// TwinCAT 3 PLC project AW_PLC
// ProgramVersion: 3.1.4023.0
// libraries:
//   Tc2_EtherCAT, * (Beckhoff Automation GmbH)
//   Tc2_Standard, * (Beckhoff Automation GmbH)
//   Tc2_System, * (Beckhoff Automation GmbH)
//   Tc3_Module, * (Beckhoff Automation GmbH)
// project tree:
//   DUTs/ TextList.TcTLO
//   / Gestore di visualizzazione.TcVMO (not stored), GlobalTextList.TcGTLO, PlcTask.TcTTO, Sfondo.TcIPO (not stored)
//   GVLs/ CONST.TcGVL, CTRL.TcGVL, ENC.TcGVL, MODE.TcGVL, MOTOR.TcGVL, PLC_ERROR.TcGVL, TRAJ.TcGVL
//   POUs/ HMI.TcPOU, INIT.TcPOU, MAIN.TcPOU, SDO.TcPOU, STATE_MACHINE.TcPOU
//   POUs/Modes/ Cyclic_sync_pos.TcPOU, Cyclic_sync_torq.TcPOU, Cyclic_sync_vel.TcPOU, Position_profile.TcPOU, Torque_profile.TcPOU, Velocity_profile.TcPOU
//   POUs/Trajectories/ BWPoly3.TcPOU, BWPoly4.TcPOU, BWPoly5.TcPOU, FWPoly3.TcPOU, FWPoly4.TcPOU, FWPoly5.TcPOU
//   VISUs/ ControlPanel.TcVIS

CONFIGURATION AW_PLC
    RESOURCE PLC ON TwinCAT3
        TASK PlcTask(INTERVAL := T#1ms, PRIORITY := 20);
        PROGRAM MAIN WITH PlcTask : MAIN;
    END_RESOURCE
END_CONFIGURATION

// ---- GVLs/CONST.TcGVL
{attribute 'qualified_only'}
VAR_GLOBAL CONSTANT
	
END_VAR
VAR_GLOBAL CONSTANT
	PI_2_MIL: DINT := 6283185;
	COUNT: DINT := 1048576;
END_VAR

// ---- GVLs/CTRL.TcGVL
{attribute 'qualified_only'}
VAR_GLOBAL
	state_axis: INT;
	working_counter_status AT %I*: BYTE;
	error AT %I*: INT;
	start					: BOOL := FALSE; 		// Start al movimento
	stop					: BOOL := FALSE;		// Stop al movimento
	opmode AT%Q*		 	: SINT := 8; 			// Modo operativo
	in_opmode AT%I* 		: SINT; 				// Modo operativo letto da giunto
	status_word AT %I*: UINT;
	control_word AT %Q*: UINT;
	sdo: BOOL := FALSE;
	a: BOOL := TRUE;
	b: BOOL;
	read_error: BOOL;
	set_up: BOOL := TRUE;
	wait: BOOL := TRUE;
	active: BOOL := TRUE;
END_VAR

// ---- GVLs/ENC.TcGVL
{attribute 'qualified_only'}
VAR_GLOBAL
		// Approssimato da 2^20/360
	DEG_TO_INC: DINT := 2912;
	RPM_TO_INCS: DINT := 17476;
END_VAR

// ---- GVLs/MODE.TcGVL
{attribute 'qualified_only'}
VAR_GLOBAL CONSTANT
	PROFILE_POSITION	: SINT := 1;
	PROFILE_VELOCITY	: SINT := 3;
	TORQUE_PROFILE		: SINT := 4;
	CYCLIC_SYNC_POS		: SINT := 8;
	CYCLIC_SYNC_VEL		: SINT := 9;
	CYCLIC_SYNC_TORQ	: SINT := 10;
END_VAR

// ---- GVLs/MOTOR.TcGVL
{attribute 'qualified_only'}
VAR_GLOBAL
END_VAR
VAR_GLOBAL
	GEAR_RATIO				: DINT 	:= 51;
	NOMINAL_CURRENT			: INT 	:= 38;	// [A]
	TORQUE_CONSTANT			: INT 	:= 115; // [mNm/A]
	actual_vel_rpm AT %I*			: DINT;		// 
	// In per thousand of the nominal torque
	actual_torque AT %I*			: INT;
	actual_pos_inc AT %I*	: DINT; 		// Posizione reale [cnt]
	RATED_TORQUE_NM: LREAL := 3;
	RATED_SPEED_RPM: UDINT := 1400;
END_VAR

// ---- GVLs/PLC_ERROR.TcGVL
{attribute 'qualified_only'}
VAR_GLOBAL CONSTANT
END_VAR
VAR_GLOBAL CONSTANT
	TRAJ_NO_SETUP: UINT := 1;
	MODE_NO_SETUP: INT := 2;
END_VAR

// ---- GVLs/TRAJ.TcGVL
{attribute 'qualified_only'}
VAR_GLOBAL
	end_pos_inc					: DINT := 0; 		// Posizione finale
	target_pos_inc AT %Q* 	: DINT; 			// Posizione target [cnt]
	// Velocità target [cnt]
	target_vel_mrpm AT %Q*	: DINT;
	start_pos_inc				: DINT := 0; 		// Posizione di start
	tempo					: LREAL := 0; 		// tempo [ms]
	offset_inc: DINT;
	periodo_ms					: LREAL := 1; 		// Durata poly5 [s]	
	delta_t					: LREAL; 			// Delta t per ogni ciclo
	v_max_incs					: DINT; 	// Velocità massima raggiungibile 
	status: BOOL := 0;
	error: UINT := 0;
	v_max_rpm_low: LREAL;
	
	position_selector_deg				: DINT := 180; 	// Offset posizione poly5 [deg]
	target_torque_per_thousand AT %Q*: INT;
	speed_selector_rpm					: UDINT := 500; 	// Velocità massima raggiungibile a freddo 1600 [rpm]
	// [Nm]
	torque_selector_Nm: LREAL := 0.40;
	speed_demand_value AT %I*: DINT;
END_VAR

// ---- POUs/MAIN.TcPOU
PROGRAM MAIN

HMI();
SDO();
STATE_MACHINE();

END_PROGRAM

// ---- POUs/HMI.TcPOU
PROGRAM HMI
VAR
	no_ecat_light: BOOL;
	error_light: BOOL;
	reset_button: BOOL;
	actual_speed_rpm: LREAL;
	actual_torque_nm_fast: LREAL;
	actual_torque_nm_slow: LREAL;
	target_error: DINT;
	count: UDINT := 0;
	status_light: BOOL;
	reset_light: BOOL;
	out_limits_light: BOOL;
	error_output: STRING;
	start_light: BOOL := FALSE;
END_VAR

IF(count = 100)THEN
	//Errors Manage
	IF((CTRL.status_word AND 16#0F)= 16#8)THEN
		error_light := TRUE;
		CTRL.read_error := TRUE;
		IF(CTRL.status_word = 16#B8)THEN
			reset_light		:= TRUE;
		END_IF
		IF(CTRL.status_word = 16#1038)THEN
			out_limits_light	:= TRUE;
		ELSE
			out_limits_light	:= FALSE;
		END_IF
	END_IF
	
	IF (CTRL.working_counter_status = 0) THEN
		no_ecat_light := FALSE;
	ELSE
		no_ecat_light := TRUE;
	END_IF
	
	IF(STATE_MACHINE.timer.Q)THEN 
		CTRL.wait := FALSE;
	ELSE
		CTRL.wait := TRUE;
	END_IF
	
	IF (NOT(CTRL.error = 0 AND TRAJ.error = 0)) THEN 
		error_light := TRUE;
	ELSE
		error_light := FALSE;
	END_IF
	
	IF(CTRL.status_word.0 = 0)THEN
		status_light := FALSE;
		CTRL.read_error := TRUE;
	ELSE
		status_light := TRUE;
		CTRL.read_error := FALSE;	
	END_IF
	
	//Buttons manager
	IF (reset_button) THEN
		STATE_MACHINE.timer(IN:=FALSE);
		CTRL.state_axis	:= 0;
		CTRL.error		:= 0;
		CTRL.control_word := 16#80;
		CTRL.sdo		:= FALSE;
		error_light 	:= FALSE;
		reset_light		:= FALSE;
		out_limits_light:= FALSE;
		reset_button 	:= FALSE;
	END_IF
	
	IF(CTRL.set_up = FALSE)THEN
		INIT();
		CTRL.state_axis	:= 0;
		CTRL.active 	:= TRUE;
	ELSE
		CTRL.active 	:= FALSE;	
	END_IF
		
	//Updates
	actual_speed_rpm		:= MOTOR.actual_vel_rpm*MOTOR.GEAR_RATIO/1000;	
	actual_torque_nm_fast 	:= (MOTOR.actual_torque * MOTOR.RATED_TORQUE_NM)/1000;
	actual_torque_nm_slow 	:= actual_torque_nm_fast * DINT_TO_LREAL(MOTOR.GEAR_RATIO);
	
	count := 0;
ELSE
	count:= count + 1;
END_IF

END_PROGRAM

// ---- POUs/STATE_MACHINE.TcPOU
PROGRAM STATE_MACHINE
VAR
	timer: TON;
END_VAR

IF ( CTRL.sdo = TRUE)THEN
	timer(IN:=TRUE);
	IF (timer.Q = TRUE) THEN
		CASE CTRL.in_opmode OF
			MODE.PROFILE_POSITION:
				Position_profile();	
			MODE.PROFILE_VELOCITY:
				Velocity_profile();
			MODE.TORQUE_PROFILE:
				Torque_profile();
			MODE.CYCLIC_SYNC_POS:
				Cyclic_sync_pos();
			MODE.CYCLIC_SYNC_VEL:
				Cyclic_sync_vel();
			MODE.CYCLIC_SYNC_TORQ:
				Cyclic_sync_torq();	
		ELSE
			CTRL.error:= PLC_ERROR.MODE_NO_SETUP;		
		END_CASE	
	END_IF
END_IF

END_PROGRAM

// ---- POUs/SDO.TcPOU
PROGRAM SDO
VAR
	
	userNetId             	: T_AmsNetId 		:= '192.168.12.90.4.1'; 	// Have to be entered
   	userSlaveAddr         	: UINT 				:= 1001;     				// Have to be entered
	//CoE reading 
	fb_coe_read1           	: FB_EcCoESdoRead;  						// Function Block for reading from CoE
	fb_coe_read2           	: FB_EcCoESdoRead;
	fb_coe_read3           	: FB_EcCoESdoRead;
	fb_coe_read4           	: FB_EcCoESdoRead;
	fb_coe_read5           	: FB_EcCoESdoRead;
	fb_coe_read6           	: FB_EcCoESdoRead;
	fb_coe_read7           	: FB_EcCoESdoRead;
	fb_coe_read8           	: FB_EcCoESdoRead;
	
	fb_coe_write1           : FB_EcCoESdoWrite;
	fb_coe_write2           : FB_EcCoESdoWrite;
	fb_coe_write3           : FB_EcCoESdoWrite;
	fb_coe_write4           : FB_EcCoESdoWrite;
	fb_coe_write5           : FB_EcCoESdoWrite;
	fb_coe_write6           : FB_EcCoESdoWrite;
	fb_coe_write7           : FB_EcCoESdoWrite;
	fb_coe_write8           : FB_EcCoESdoWrite;
	fb_coe_write9           : FB_EcCoESdoWrite;
	fb_coe_write10          : FB_EcCoESdoWrite;
	fb_coe_write11          : FB_EcCoESdoWrite;
	fb_coe_write12          : FB_EcCoESdoWrite;
	fb_coe_write13          : FB_EcCoESdoWrite;
	fb_coe_write14          : FB_EcCoESdoWrite;
	
	motor_revolutions		: UDINT;
	shaft_revolutions		: UDINT;
	enc_resolution			: UDINT := 1048576;
	motor_rated_torque		: DINT;
	max_motor_speed			: UDINT;	
	
	profile_velocity		: UDINT := 0;
	profile_acceleration	: UDINT := 20000;
	profile_deceleration	: UDINT := 20000;
	quick_stop_deceleration	: UDINT := 10000;
	position_window			: UDINT := 100;
	velocity_window			: UINT := 500;
	velocity_window_time	: UINT := 0;
	torque_window			: UINT := 100;
	torque_window_time		: UINT := 0;
	torque_slope			: UDINT := 100;
	written_speed			: UDINT;
	count: INT := 0;
	bExecuteworld: BOOL := FALSE;
	error_report: STRING;
	position_filter_type: USINT := 1;
	position_filter_frequency: UDINT := 200;
	r_position_filter_type: USINT;
	r_position_filter_frequency: UDINT;
	velocity_filter_type: USINT := 1;
	velocity_filter_frequency: UDINT := 100;
END_VAR

//****************** SDO *****************
IF (CTRL.read_error = TRUE) THEN
	fb_coe_read6(bExecute := FALSE);
	fb_coe_read6(
			sNetId		:= userNetId, 
			nSlaveAddr	:= userSlaveAddr, 
			nSubIndex	:= 1, 
			nIndex		:= 16#203F,
			pDstBuf		:= ADR(error_report), 
			cbBufLen    := SIZEOF(error_report), 
			bExecute    := TRUE, 
			tTimeout    := T#1S);
	CTRL.read_error := FALSE;
END_IF

IF (CTRL.sdo = FALSE AND HMI.error_light = FALSE)  THEN

    // read
	IF ( count = 0 ) THEN
		fb_coe_read1(bExecute := FALSE);
		fb_coe_read2(bExecute := FALSE);
		fb_coe_read3(bExecute := FALSE);
		fb_coe_read4(bExecute := FALSE);
		fb_coe_read5(bExecute := FALSE);
		fb_coe_write1(bExecute := FALSE);
		fb_coe_write2(bExecute := FALSE);
		fb_coe_write3(bExecute := FALSE);
		fb_coe_write4(bExecute := FALSE);
		fb_coe_write5(bExecute := FALSE);
		fb_coe_write6(bExecute := FALSE);
		fb_coe_write7(bExecute := FALSE);
		fb_coe_write8(bExecute := FALSE);
		fb_coe_write9(bExecute := FALSE);
		fb_coe_write10(bExecute := FALSE);
		fb_coe_write11(bExecute := FALSE);
		fb_coe_write12(bExecute := FALSE);
		fb_coe_write13(bExecute := FALSE);
		fb_coe_write14(bExecute := FALSE);
		count := count +1;
		STATE_MACHINE.timer(IN:=FALSE,PT:=T#4S);
	END_IF

	
	IF ( NOT bExecuteworld AND count = 1) THEN
		fb_coe_read1(
			sNetId        := userNetId, 
			nSlaveAddr    := userSlaveAddr, 
			nSubIndex    := 1, 
			nIndex        := 16#6091,
			pDstBuf        := ADR(motor_revolutions), 
			cbBufLen    := SIZEOF(motor_revolutions), 
			bExecute    := TRUE, 
			tTimeout    := T#1S);
	
		IF (NOT fb_coe_read1.bBusy) THEN
			bExecuteworld := FALSE;
			fb_coe_read1(bExecute := FALSE);
			count := count + 1;
		END_IF
		
	END_IF
	IF ( NOT bExecuteworld AND count = 2) THEN
		fb_coe_read2(
			sNetId        := userNetId, 
			nSlaveAddr    := userSlaveAddr, 
			nSubIndex    := 2, 
			nIndex        := 16#6091,
			pDstBuf     := ADR(shaft_revolutions), 
			cbBufLen    := SIZEOF(shaft_revolutions), 
			bExecute    := TRUE, 
			tTimeout    := T#1S);	
			
		IF (NOT fb_coe_read2.bBusy) THEN
			bExecuteworld := FALSE;
			fb_coe_read2(bExecute := FALSE);
			count := count + 1;
		END_IF
		
	END_IF
	IF ( NOT bExecuteworld AND count = 3) THEN
		fb_coe_read3(
			sNetId        := userNetId, 
			nSlaveAddr    := userSlaveAddr, 
			nSubIndex    := 3, 
			nIndex        := 16#2110,
			pDstBuf        := ADR(enc_resolution), 
			cbBufLen    := SIZEOF(enc_resolution), 
			bExecute    := TRUE, 
			tTimeout    := T#1S);
	
		IF (NOT fb_coe_read3.bBusy) THEN
			bExecuteworld := FALSE;
			fb_coe_read3(bExecute := FALSE);
			count := count + 1;
		END_IF
		
	END_IF
	IF ( NOT bExecuteworld AND count = 4) THEN
		fb_coe_read4(
			sNetId      := userNetId, 
			nSlaveAddr  := userSlaveAddr, 
			nSubIndex   := 0, 
			nIndex      := 16#6076,
			pDstBuf     := ADR(motor_rated_torque), 
			cbBufLen    := SIZEOF(motor_rated_torque), 
			bExecute    := TRUE, 
			tTimeout    := T#1S);
		IF (NOT fb_coe_read4.bBusy) THEN
			bExecuteworld := FALSE;
			fb_coe_read4(bExecute := FALSE);
			count := count + 1;
		END_IF
		
	END_IF
	IF ( NOT bExecuteworld AND count = 5) THEN
		fb_coe_read5(
			sNetId      := userNetId, 
			nSlaveAddr  := userSlaveAddr, 
			nSubIndex   := 0, 
			nIndex      := 16#6080,
			pDstBuf     := ADR(max_motor_speed), 
			cbBufLen    := SIZEOF(max_motor_speed), 
			bExecute    := TRUE, 
			tTimeout    := T#1S);
		IF (NOT fb_coe_read5.bBusy) THEN
			bExecuteworld := FALSE;
			fb_coe_read5(bExecute := FALSE);
			count := count + 1;
		END_IF
	END_IF
	IF ( NOT bExecuteworld AND count = 6) THEN
		fb_coe_read7(
			sNetId      := userNetId, 
			nSlaveAddr  := userSlaveAddr, 
			nSubIndex   := 1, 
			nIndex      := 16#2022,
			pDstBuf     := ADR(r_position_filter_type), 
			cbBufLen    := SIZEOF(r_position_filter_type), 
			bExecute    := TRUE, 
			tTimeout    := T#1S);
		IF (NOT fb_coe_read7.bBusy) THEN
			bExecuteworld := FALSE;
			fb_coe_read7(bExecute := FALSE);
			count := count + 1;
		END_IF
	END_IF
	IF ( NOT bExecuteworld AND count = 7) THEN
		fb_coe_read8(
			sNetId      := userNetId, 
			nSlaveAddr  := userSlaveAddr, 
			nSubIndex   := 2, 
			nIndex      := 16#2022,
			pDstBuf     := ADR(r_position_filter_frequency), 
			cbBufLen    := SIZEOF(r_position_filter_frequency), 
			bExecute    := TRUE, 
			tTimeout    := T#1S);
		IF (NOT fb_coe_read8.bBusy) THEN
			bExecuteworld := FALSE;
			fb_coe_read8(bExecute := FALSE);
			count := count + 1;
		END_IF
	END_IF
	
    //write
	
	IF ( NOT bExecuteworld AND count = 8) THEN
		//defined by user panel
		profile_velocity 	:= TRAJ.speed_selector_rpm * 1000/DINT_TO_UDINT(MOTOR.GEAR_RATIO);
		fb_coe_write1(
			sNetId     := userNetId,
			nSlaveAddr := userSlaveAddr,
			nIndex     := 16#6081,
			nSubIndex  := 0,
			pSrcBuf    := ADR(profile_velocity),
			cbBufLen   := SIZEOF(profile_velocity),
			bExecute   := TRUE);
		IF (NOT fb_coe_write1.bBusy) THEN
			bExecuteworld := FALSE;
			fb_coe_write1(bExecute := FALSE);
			count := count + 1;
		END_IF
	END_IF
	IF ( NOT bExecuteworld AND count = 9) THEN
		fb_coe_write2(
			sNetId     := userNetId,
			nSlaveAddr := userSlaveAddr,
			nIndex     := 16#6083,
			nSubIndex  := 0,
			pSrcBuf    := ADR(profile_acceleration),
			cbBufLen   := SIZEOF(profile_acceleration),
			bExecute   := TRUE);
		IF (NOT fb_coe_write2.bBusy) THEN
			bExecuteworld := FALSE;
			fb_coe_write2(bExecute := FALSE);
			count := count + 1;
		END_IF
	END_IF
	IF ( NOT bExecuteworld AND count = 10) THEN
		fb_coe_write3(
			sNetId     := userNetId,
			nSlaveAddr := userSlaveAddr,
			nIndex     := 16#6084,
			nSubIndex  := 0,
			pSrcBuf    := ADR(profile_deceleration),
			cbBufLen   := SIZEOF(profile_deceleration),
			bExecute   := TRUE);
		IF (NOT fb_coe_write3.bBusy) THEN
			bExecuteworld := FALSE;
			fb_coe_write3(bExecute := FALSE);
			count := count + 1;
		END_IF
	END_IF
	IF ( NOT bExecuteworld AND count = 11) THEN
		fb_coe_write4(
			sNetId     := userNetId,
			nSlaveAddr := userSlaveAddr,
			nIndex     := 16#6085,
			nSubIndex  := 0,
			pSrcBuf    := ADR(quick_stop_deceleration),
			cbBufLen   := SIZEOF(quick_stop_deceleration),
			bExecute   := TRUE);
		IF (NOT fb_coe_write4.bBusy) THEN
			bExecuteworld := FALSE;
			fb_coe_write4(bExecute := FALSE);
			count := count + 1;
		END_IF
	END_IF
	IF ( NOT bExecuteworld AND count = 12) THEN
		fb_coe_write5(
			sNetId     := userNetId,
			nSlaveAddr := userSlaveAddr,
			nIndex     := 16#6067,
			nSubIndex  := 0,
			pSrcBuf    := ADR(position_window),
			cbBufLen   := SIZEOF(position_window),
			bExecute   := TRUE);
		IF (NOT fb_coe_write5.bBusy) THEN
			bExecuteworld := FALSE;
			fb_coe_write5(bExecute := FALSE);
			count := count + 1;
		END_IF
	END_IF
	IF ( NOT bExecuteworld AND count = 13) THEN
		fb_coe_write6(
			sNetId     := userNetId,
			nSlaveAddr := userSlaveAddr,
			nIndex     := 16#606D,
			nSubIndex  := 0,
			pSrcBuf    := ADR(velocity_window),
			cbBufLen   := SIZEOF(velocity_window),
			bExecute   := TRUE);
		IF (NOT fb_coe_write6.bBusy) THEN
			bExecuteworld := FALSE;
			fb_coe_write6(bExecute := FALSE);
			count := count + 1;
		END_IF
	END_IF
	IF ( NOT bExecuteworld AND count = 14) THEN
		fb_coe_write7(
			sNetId     := userNetId,
			nSlaveAddr := userSlaveAddr,
			nIndex     := 16#606E,
			nSubIndex  := 0,
			pSrcBuf    := ADR(velocity_window_time),
			cbBufLen   := SIZEOF(velocity_window_time),
			bExecute   := TRUE);
		IF (NOT fb_coe_write7.bBusy) THEN
			bExecuteworld := FALSE;
			fb_coe_write7(bExecute := FALSE);
			count := count + 1;
		END_IF
	END_IF
	IF ( NOT bExecuteworld AND count = 15) THEN
		fb_coe_write8(
			sNetId     := userNetId,
			nSlaveAddr := userSlaveAddr,
			nIndex     := 16#2014,
			nSubIndex  := 1,
			pSrcBuf    := ADR(torque_window),
			cbBufLen   := SIZEOF(torque_window),
			bExecute   := TRUE);
		IF (NOT fb_coe_write8.bBusy) THEN
			bExecuteworld := FALSE;
			fb_coe_write8(bExecute := FALSE);
			count := count + 1;
		END_IF
	END_IF
	IF ( NOT bExecuteworld AND count = 16) THEN
		fb_coe_write9(
			sNetId     := userNetId,
			nSlaveAddr := userSlaveAddr,
			nIndex     := 16#2014,
			nSubIndex  := 2,
			pSrcBuf    := ADR(torque_window_time),
			cbBufLen   := SIZEOF(torque_window_time),
			bExecute   := TRUE);
		IF (NOT fb_coe_write9.bBusy) THEN
			bExecuteworld := FALSE;
			fb_coe_write9(bExecute := FALSE);
			count := count + 1;
		END_IF
	END_IF
	IF ( NOT bExecuteworld AND count = 17) THEN
		fb_coe_write10(
			sNetId     := userNetId,
			nSlaveAddr := userSlaveAddr,
			nIndex     := 16#6087,
			nSubIndex  := 0,
			pSrcBuf    := ADR(torque_slope),
			cbBufLen   := SIZEOF(torque_slope),
			bExecute   := TRUE);
		IF (NOT fb_coe_write10.bBusy) THEN
			bExecuteworld := FALSE;
			fb_coe_write10(bExecute := FALSE);
			count := count + 1;
		END_IF		
	END_IF
	IF ( NOT bExecuteworld AND count = 18) THEN
		fb_coe_write11(
			sNetId     := userNetId,
			nSlaveAddr := userSlaveAddr,
			nIndex     := 16#2022,
			nSubIndex  := 1,
			pSrcBuf    := ADR(position_filter_type),
			cbBufLen   := SIZEOF(position_filter_type),
			bExecute   := TRUE);
		IF (NOT fb_coe_write11.bBusy) THEN
			bExecuteworld := FALSE;
			fb_coe_write11(bExecute := FALSE);
			count := count + 1;
		END_IF		
	END_IF
	IF ( NOT bExecuteworld AND count = 19) THEN
		fb_coe_write12(
			sNetId     := userNetId,
			nSlaveAddr := userSlaveAddr,
			nIndex     := 16#2022,
			nSubIndex  := 2,
			pSrcBuf    := ADR(position_filter_frequency),
			cbBufLen   := SIZEOF(position_filter_frequency),
			bExecute   := TRUE);
		IF (NOT fb_coe_write12.bBusy) THEN
			bExecuteworld := FALSE;
			fb_coe_write12(bExecute := FALSE);
			count := count + 1;
		END_IF		
	END_IF
	IF ( NOT bExecuteworld AND count = 20) THEN
		fb_coe_write13(
			sNetId     := userNetId,
			nSlaveAddr := userSlaveAddr,
			nIndex     := 16#2021,
			nSubIndex  := 1,
			pSrcBuf    := ADR(velocity_filter_type),
			cbBufLen   := SIZEOF(velocity_filter_type),
			bExecute   := TRUE);
		IF (NOT fb_coe_write13.bBusy) THEN
			bExecuteworld := FALSE;
			fb_coe_write13(bExecute := FALSE);
			count := count + 1;
		END_IF		
	END_IF
	IF ( NOT bExecuteworld AND count = 21) THEN
		fb_coe_write14(
			sNetId     := userNetId,
			nSlaveAddr := userSlaveAddr,
			nIndex     := 16#2021,
			nSubIndex  := 2,
			pSrcBuf    := ADR(velocity_filter_frequency),
			cbBufLen   := SIZEOF(velocity_filter_frequency),
			bExecute   := TRUE);
		IF (NOT fb_coe_write14.bBusy) THEN
			bExecuteworld := FALSE;
			fb_coe_write14(bExecute := FALSE);
			CTRL.sdo     := TRUE;
			count := 0;
		END_IF		
	END_IF		
END_IF

END_PROGRAM

// ---- POUs/Modes/Position_profile.TcPOU
PROGRAM Position_profile
VAR
	back: BOOL := TRUE;
	timer_test: TON;
	timer_bool: BOOL := FALSE;
	
	fb_coe_write           : FB_EcCoESdoWrite;
	profile_velocity: UDINT := 0;
END_VAR

//PROFILE POSITION MODE
CASE CTRL.state_axis OF

	0:
		IF (CTRL.start AND timer_bool = FALSE) THEN	
			timer_test(IN:=FALSE,PT:=T#3S);
			timer_bool := TRUE;
			fb_coe_write(bExecute := FALSE);
			INIT();	
		ELSE
			IF (CTRL.start) THEN
				profile_velocity 	:= TRAJ.speed_selector_rpm * 1000/DINT_TO_UDINT(MOTOR.GEAR_RATIO);
				fb_coe_write(
					sNetId     := SDO.userNetId,
					nSlaveAddr := SDO.userSlaveAddr,
					nIndex     := 16#6081,
					nSubIndex  := 0,
					pSrcBuf    := ADR(profile_velocity),
					cbBufLen   := SIZEOF(profile_velocity),
					bExecute   := TRUE);

				IF(timer_bool = TRUE) THEN
					//fb_coe_write(bExecute := FALSE);
					IF (NOT fb_coe_write.bBusy) THEN
						timer_test(IN:=TRUE);
						IF ( timer_test.Q = TRUE ) THEN
							CTRL.start		:= FALSE;
							CTRL.state_axis	:= 5;
							timer_bool 		:= FALSE;  
						END_IF		
					END_IF	
				END_IF
			END_IF
		END_IF
	
    5: // State 5: Switch on request
		IF (timer_bool = FALSE) THEN
			CTRL.control_word       := 16#6;        // Reset status
			TRAJ.target_pos_inc     := MOTOR.actual_pos_inc;
			timer_test(IN:=FALSE,PT:=T#3S);
			IF ((CTRL.status_word.0 = 1) AND (CTRL.status_word.4 = 1) AND (CTRL.error = 0)) THEN
				CTRL.control_word	:= 16#7;        // Switch on
				TRAJ.target_pos_inc	:= MOTOR.actual_pos_inc;	
				timer_bool := TRUE;
			END_IF
		ELSE
			timer_test(IN:=TRUE);
			IF ( timer_test.Q = TRUE ) THEN
				CTRL.state_axis	:= 10;
				timer_bool 		:= FALSE;  
			END_IF
		END_IF
					
    10: // State 20: verify operation enable flag and that the operation mode is correctly set on the driver
		IF (timer_bool = FALSE) THEN
			IF ((CTRL.error = 0) AND (CTRL.status_word.1 = 1) AND (CTRL.in_opmode = MODE.PROFILE_POSITION)) THEN
				CTRL.start		:= FALSE;
				TRAJ.offset_inc	:= (TRAJ.position_selector_deg * ENC.DEG_TO_INC);
				IF( back = TRUE) THEN
					TRAJ.target_pos_inc	:= 0;
					back				:= FALSE;
				ELSE
					TRAJ.target_pos_inc	:= TRAJ.offset_inc;
					back				:= TRUE;
				END_IF
				//CTRL.control_word.3     := 1; // operation enable
				CTRL.control_word := 16#0F;
				timer_test(IN:=FALSE,PT:=T#3S);
				timer_bool := TRUE;
			END_IF
		ELSE
			timer_test(IN:=TRUE);
			IF ( timer_test.Q = TRUE ) THEN
				CTRL.state_axis	:= 15;
				timer_bool		:= FALSE;  
			END_IF
		END_IF
	
	15:
		IF (timer_bool = FALSE) THEN
			CTRL.control_word := 16#3F;
			//CTRL.control_word.4     := 1; // new set-point
			//CTRL.control_word.5     := 1; // change set immediately
			timer_test(IN:=FALSE,PT:=T#1S);
			timer_bool := TRUE;
		ELSE
			timer_test(IN:=TRUE);
			IF ( timer_test.Q = TRUE ) THEN
				CTRL.state_axis	:= 20;
				timer_bool		:= FALSE;  
			END_IF
		END_IF

    20: // State 30: verify the set-point acknowledge
        IF ((CTRL.error = 0)  AND (CTRL.status_word.12 = 1)) THEN
            CTRL.state_axis         := 30;
        END_IF

    30: // State 40: wait target reached and swap target position
        IF ( CTRL.status_word.10 = 1 ) THEN
            IF (CTRL.stop) THEN
                CTRL.state_axis     := 40;
                back                := FALSE;
            ELSE
                CTRL.state_axis     := 10;
            END_IF
//This section has been commented out due to errors and a subsequently reset after sudden stops.
//		ELSE 
//			IF (CTRL.stop) THEN
//				CTRL.state_axis     := 40;
//                back                := FALSE;
//			END_IF
        END_IF

    40: // State 50: switch off request
        CTRL.control_word	:= 0; 
        CTRL.start			:= 0;
        CTRL.stop			:= 0;
        CTRL.state_axis		:= 0;
END_CASE

END_PROGRAM

// ---- POUs/INIT.TcPOU
PROGRAM INIT

VAR
	once: BOOL := FALSE;
END_VAR

IF(once=FALSE)THEN
	ENC.DEG_TO_INC := UDINT_TO_DINT(SDO.enc_resolution/360);
	ENC.RPM_TO_INCS:= UDINT_TO_DINT(SDO.enc_resolution/60);
	MOTOR.GEAR_RATIO := UDINT_TO_DINT(SDO.motor_revolutions/SDO.shaft_revolutions);
	MOTOR.RATED_TORQUE_NM 	:= DINT_TO_LREAL(SDO.motor_rated_torque)/1000.0;	
	MOTOR.RATED_SPEED_RPM	:= SDO.max_motor_speed/1000;
	once := TRUE;
END_IF

END_PROGRAM

// ---- POUs/Modes/Velocity_profile.TcPOU
PROGRAM Velocity_profile

VAR
	v_max_mrpm: DINT;
	back: BOOL := TRUE;
	timer_test: TON;
	timer_bool: BOOL := FALSE;
	fb_coe_write: INT;
	profile_velocity: DINT;
END_VAR

// PROFILE VELOCITY MODE
CASE CTRL.state_axis OF

    0: // State 0: Switch on request
		IF (timer_bool = FALSE) THEN
			CTRL.control_word	:= 16#6;        // Reset status
			TRAJ.target_vel_mrpm := 0;
			timer_test(IN:=FALSE,PT:=T#3S);
			IF ((CTRL.status_word.0 = 1) AND (CTRL.status_word.4 = 1) AND (CTRL.error = 0) AND CTRL.start) THEN
				CTRL.control_word	:= 16#7;        // Switch on
				INIT();
				timer_bool := TRUE;
			END_IF
		ELSE
			IF (timer_bool)THEN
				timer_test(IN:=TRUE);
				IF ( timer_test.Q = TRUE ) THEN
					CTRL.start		:= FALSE;
					CTRL.state_axis	:= 10;
					timer_bool 		:= FALSE;  
				END_IF
			END_IF
		END_IF
        
    10: // State 10: verify operation enable flag and that the operation mode is correctly set on the driver
		IF(timer_bool = FALSE) THEN
			IF ((CTRL.error = 0) AND (CTRL.status_word.1 = 1) AND (CTRL.in_opmode = MODE.PROFILE_VELOCITY)) THEN           
				v_max_mrpm 	:= UDINT_TO_DINT(TRAJ.speed_selector_rpm * 1000)/MOTOR.GEAR_RATIO;
				IF( back = TRUE) THEN
					TRAJ.target_vel_mrpm    := - v_max_mrpm;
					back                    := FALSE;
				ELSE
					TRAJ.target_vel_mrpm    := v_max_mrpm;
					back                    := TRUE;
				END_IF
				//CTRL.control_word.3     := 1; // operation enable
				CTRL.control_word := 16#0F;
				timer_test(IN:=FALSE,PT:=T#3S);
				timer_bool := TRUE;
			END_IF
		ELSE
			timer_test(IN:=TRUE);
			IF ( timer_test.Q = TRUE ) THEN
				CTRL.state_axis	:= 20;
				timer_bool		:= FALSE;  
			END_IF			
		END_IF
		
    20: // State 20: wait target reached and swap target profile
        IF ( CTRL.status_word.10 = 1 ) THEN
            IF (CTRL.stop) THEN
                CTRL.state_axis     := 30;
                back                := FALSE;
            ELSE
                CTRL.state_axis     := 10;
                CTRL.status_word.8  := 1; // halt flag on
            END_IF
        END_IF

    30: // State 30: switch off request 
        CTRL.start			:= 0;
        CTRL.stop			:= 0;
		TRAJ.target_vel_mrpm:= 0;
		IF(ABS(MOTOR.actual_vel_rpm) < SDO.velocity_window)THEN
			CTRL.control_word	:= 0;
        	CTRL.state_axis		:= 0;
		END_IF
END_CASE

END_PROGRAM

// ---- POUs/Modes/Torque_profile.TcPOU
PROGRAM Torque_profile
VAR
	back: BOOL;
	torque_per_thousand: INT;
	timer_bool: BOOL := FALSE;
	timer_test: TON;
END_VAR

//PROFILE TORQUE MODE
CASE CTRL.state_axis OF
	
    0: // State 0: Switch on request
		IF (timer_bool = FALSE) THEN
			CTRL.control_word	:= 16#6;        // Reset status
			TRAJ.target_torque_per_thousand := 0;
			timer_test(IN:=FALSE,PT:=T#3S);
			IF ((CTRL.status_word.0 = 1) AND (CTRL.status_word.4 = 1) AND (CTRL.error = 0) AND CTRL.start) THEN
				CTRL.control_word	:= 16#7;        // Switch on
				INIT();
				timer_bool := TRUE;
			END_IF
		ELSE
			IF (timer_bool)THEN
				timer_test(IN:=TRUE);
				IF ( timer_test.Q = TRUE ) THEN
					CTRL.start		:= FALSE;
					CTRL.state_axis	:= 10;
					timer_bool 		:= FALSE;  
				END_IF
			END_IF
		END_IF

    10: // State 10: verify operation enable flag and that the operation mode is correctly set on the driver
		IF(timer_bool = FALSE) THEN
			IF ((CTRL.error = 0) AND (CTRL.status_word.1 = 1) AND (CTRL.in_opmode = MODE.TORQUE_PROFILE)) THEN          
				torque_per_thousand := LREAL_TO_INT((TRAJ.torque_selector_Nm*1000)/MOTOR.RATED_TORQUE_NM);
				IF( back = TRUE) THEN
					TRAJ.target_torque_per_thousand    := -torque_per_thousand;
					back                     := FALSE;
				ELSE
					TRAJ.target_torque_per_thousand    := torque_per_thousand;
					back                     := TRUE;
				END_IF
				//CTRL.control_word.3     := 1; // operation enable
				CTRL.control_word := 16#0F;
				timer_test(IN:=FALSE,PT:=T#3S);
				timer_bool := TRUE;
			END_IF
		ELSE
			timer_test(IN:=TRUE);
			IF ( timer_test.Q = TRUE ) THEN
				CTRL.state_axis	:= 20;
				timer_bool		:= FALSE;  
			END_IF			
		END_IF		
			
    20: // State 20: wait target reached and swap target position
        IF ( CTRL.status_word.10 = 1 ) THEN
            IF (CTRL.stop) THEN
                CTRL.state_axis     := 30;
                back                 := FALSE;
            ELSE
                CTRL.state_axis     := 10;
                CTRL.status_word.8  := 1; // halt flag on
            END_IF
        END_IF

    30: // State 30: switch off request
        CTRL.start			:= 0;
        CTRL.stop			:= 0;
		TRAJ.target_torque_per_thousand	:= 0;
		IF(ABS(MOTOR.actual_torque) < UINT_TO_INT(SDO.torque_window))THEN
			CTRL.control_word	:= 0;
        	CTRL.state_axis		:= 0;
		END_IF
END_CASE

END_PROGRAM

// ---- POUs/Modes/Cyclic_sync_pos.TcPOU
PROGRAM Cyclic_sync_pos

VAR
	timer_bool: BOOL;
	timer_test: TON;
	back: BOOL;
END_VAR

// Macchina a stati comandi giunto
CASE CTRL.state_axis OF
	
    0: // State 0: Switch on request
		IF (timer_bool = FALSE) THEN
			CTRL.control_word	:= 16#6;        // Reset status
			
			timer_test(IN:=FALSE,PT:=T#3S);
			IF ((CTRL.status_word.0 = 1) AND (CTRL.status_word.4 = 1) AND (CTRL.error = 0) AND CTRL.start) THEN
				CTRL.control_word	:= 16#7;        // Switch on
				INIT();
				timer_bool := TRUE;
			END_IF
		ELSE
			IF (timer_bool)THEN
				timer_test(IN:=TRUE);
				IF ( timer_test.Q = TRUE ) THEN
					CTRL.start		:= FALSE;
					CTRL.state_axis	:= 10;
					timer_bool 		:= FALSE;  
				END_IF
			END_IF
		END_IF
	
    10:
		IF(timer_bool = FALSE) THEN
			IF ((CTRL.error = 0) AND (CTRL.status_word.1 = 1) AND (CTRL.in_opmode = MODE.CYCLIC_SYNC_POS)) THEN           
				TRAJ.target_pos_inc	:= MOTOR.actual_pos_inc;
				CTRL.control_word := 16#0F;
				timer_test(IN:=FALSE,PT:=T#3S);
				timer_bool := TRUE;
			END_IF
		ELSE
			timer_test(IN:=TRUE);
			IF ( timer_test.Q = TRUE ) THEN
				CTRL.state_axis	:= 20;
				timer_bool	:= FALSE;  
			END_IF			
		END_IF
		
	20:
		TRAJ.target_pos_inc	:= MOTOR.actual_pos_inc;
		IF ((CTRL.error = 0) AND (CTRL.in_opmode = MODE.CYCLIC_SYNC_POS)) THEN
			TRAJ.tempo 		:= 0;
			IF( back = TRUE) THEN
				back			:= FALSE;
				CTRL.state_axis	:= 30;
			ELSE
				back			:= TRUE;
				CTRL.state_axis	:= 40;
			END_IF
		END_IF
	
	30:
		FWPoly5();  
		IF (TRAJ.tempo >= 1) THEN
			TRAJ.status := FALSE;
			IF (CTRL.stop) THEN
				CTRL.state_axis := 50;
			ELSE
				CTRL.state_axis := 20;
			END_IF
		ELSE
			TRAJ.tempo := TRAJ.tempo + TRAJ.delta_t;
		END_IF  
         
    40:
		BWPoly5();
		IF (TRAJ.tempo >= 1) THEN
			TRAJ.status := FALSE;
			IF (CTRL.stop) THEN
				CTRL.state_axis := 50;
			ELSE
				CTRL.state_axis := 20;
			END_IF
		ELSE
			TRAJ.tempo := TRAJ.tempo + TRAJ.delta_t;
		END_IF    
               
	50:
		CTRL.control_word	:= 0; 
		CTRL.start 		:= 0;
		CTRL.stop  		:= 0;
		CTRL.state_axis := 0;                                                                                                                                                                                                                                                                                                                                                                                                                                                                                                                                                            
END_CASE

END_PROGRAM

// ---- POUs/Trajectories/FWPoly5.TcPOU
PROGRAM FWPoly5
VAR
	a						: LREAL; 			// Coefficiente "a" poly5
	b						: LREAL; 			// Coefficiente "b" poly5
	c						: LREAL; 			// Coefficiente "c" poly5
	tempo_2					: LREAL; 			// Tempo ^2
	tempo_3					: LREAL; 			// Tempo ^3
	tempo_4					: LREAL; 			// Tempo ^4
	tempo_5					: LREAL;	 		// Tempo ^5
END_VAR

IF (TRAJ.tempo = 0) THEN
	TRAJ.offset_inc		:= (TRAJ.position_selector_deg * ENC.DEG_TO_INC);
	TRAJ.v_max_rpm_low	:= (UDINT_TO_LREAL(TRAJ.speed_selector_rpm) / MOTOR.GEAR_RATIO);
	TRAJ.periodo_ms 	:= (ABS(TRAJ.position_selector_deg) * 15 * 1000) / (8 * TRAJ.v_max_rpm_low * 6) ; // millisecondi
	TRAJ.status			:= TRUE;
	TRAJ.delta_t 		:= 1 / (TRAJ.periodo_ms); 
	
	a := 6 * TRAJ.offset_inc;
	b := -15 * TRAJ.offset_inc;
	c := 10 * TRAJ.offset_inc;
	
	TRAJ.start_pos_inc := MOTOR.actual_pos_inc;
	TRAJ.end_pos_inc := (MOTOR.actual_pos_inc + TRAJ.offset_inc); 
END_IF

IF (TRAJ.status = TRUE) THEN
	tempo_2 := TRAJ.tempo * TRAJ.tempo;
	tempo_3 := tempo_2 * TRAJ.tempo;
	tempo_4 := tempo_3 * TRAJ.tempo;
	tempo_5 := tempo_4 * TRAJ.tempo;
	TRAJ.target_pos_inc := (LREAL_TO_DINT(a * tempo_5 + b * tempo_4 + c * tempo_3) + TRAJ.start_pos_inc);
ELSE
	TRAJ.error := PLC_ERROR.TRAJ_NO_SETUP;
END_IF

END_PROGRAM

// ---- POUs/Trajectories/BWPoly5.TcPOU
PROGRAM BWPoly5
VAR
	a						: LREAL; 			// Coefficiente "a" poly5
	b						: LREAL; 			// Coefficiente "b" poly5
	c						: LREAL; 			// Coefficiente "c" poly5
	tempo_2					: LREAL; 			// Tempo ^2
	tempo_3					: LREAL; 			// Tempo ^3
	tempo_4					: LREAL; 			// Tempo ^4
	tempo_5					: LREAL;	 		// Tempo ^5
END_VAR

IF (TRAJ.tempo = 0) THEN
	TRAJ.offset_inc		:= (TRAJ.position_selector_deg * ENC.DEG_TO_INC);
	TRAJ.v_max_rpm_low	:= (UDINT_TO_LREAL(TRAJ.speed_selector_rpm) / MOTOR.GEAR_RATIO);
	TRAJ.periodo_ms 	:= (ABS(TRAJ.position_selector_deg) * 15 * 1000) / (8 * TRAJ.v_max_rpm_low * 6) ; // millisecondi
	TRAJ.status			:= TRUE;
	TRAJ.delta_t 		:= 1 / (TRAJ.periodo_ms); 
	
	a := -6 * TRAJ.offset_inc;
	b := 15 * TRAJ.offset_inc;
	c := -10 * TRAJ.offset_inc;
	
	TRAJ.start_pos_inc := MOTOR.actual_pos_inc;
	TRAJ.end_pos_inc := (MOTOR.actual_pos_inc + TRAJ.offset_inc); 
END_IF

IF (TRAJ.status = TRUE) THEN
	tempo_2 := TRAJ.tempo * TRAJ.tempo;
	tempo_3 := tempo_2 * TRAJ.tempo;
	tempo_4 := tempo_3 * TRAJ.tempo;
	tempo_5 := tempo_4 * TRAJ.tempo;
	TRAJ.target_pos_inc := (LREAL_TO_DINT(a * tempo_5 + b * tempo_4 + c * tempo_3) + TRAJ.start_pos_inc);
ELSE
	TRAJ.error := PLC_ERROR.TRAJ_NO_SETUP;
END_IF

END_PROGRAM

// ---- POUs/Modes/Cyclic_sync_vel.TcPOU
PROGRAM Cyclic_sync_vel
VAR
	timer_bool: BOOL := FALSE;
	timer_test: TON;
	back: BOOL;
END_VAR

//CYCLIC SYNC VELOCITY
CASE CTRL.state_axis OF
	
    0: // State 0: Switch on request
		IF (timer_bool = FALSE) THEN
			CTRL.control_word	:= 16#6;        // Reset status
			
			timer_test(IN:=FALSE,PT:=T#3S);
			IF ((CTRL.status_word.0 = 1) AND (CTRL.status_word.4 = 1) AND (CTRL.error = 0) AND CTRL.start) THEN
				CTRL.control_word	:= 16#7;        // Switch on
				INIT();
				timer_bool := TRUE;
			END_IF
		ELSE
			IF (timer_bool)THEN
				timer_test(IN:=TRUE);
				IF ( timer_test.Q = TRUE ) THEN
					CTRL.start		:= FALSE;
					CTRL.state_axis	:= 10;
					timer_bool 		:= FALSE;  
				END_IF
			END_IF
		END_IF
	
    10:
		IF(timer_bool = FALSE) THEN
			IF ((CTRL.error = 0) AND (CTRL.status_word.1 = 1) AND (CTRL.in_opmode = MODE.CYCLIC_SYNC_VEL)) THEN           
				TRAJ.target_vel_mrpm	:= 0;
				CTRL.control_word := 16#0F;
				timer_test(IN:=FALSE,PT:=T#3S);
				timer_bool := TRUE;
			END_IF
		ELSE
			timer_test(IN:=TRUE);
			IF ( timer_test.Q = TRUE ) THEN
				CTRL.state_axis	:= 20;
				timer_bool	:= FALSE;  
			END_IF			
		END_IF
		
	20:
		TRAJ.target_vel_mrpm	:= 0;
		IF ((CTRL.error = 0) AND (CTRL.in_opmode = MODE.CYCLIC_SYNC_VEL)) THEN
			TRAJ.tempo 		:= 0;
			IF( back = TRUE) THEN
				back			:= FALSE;
				CTRL.state_axis	:= 30;
			ELSE
				back			:= TRUE;
				CTRL.state_axis	:= 40;
			END_IF
		END_IF
	
	30: 
		FWPoly4();  
		IF (TRAJ.tempo >= 1) THEN
			TRAJ.status := FALSE;
			IF (CTRL.stop) THEN
				CTRL.state_axis := 50;
			ELSE
				CTRL.state_axis := 20;
			END_IF
		ELSE
			TRAJ.tempo := TRAJ.tempo + TRAJ.delta_t;
		END_IF  
         
    40: 
		BWPoly4();
		IF (TRAJ.tempo >= 1) THEN
			TRAJ.status := FALSE;
			IF (CTRL.stop) THEN
				CTRL.state_axis := 50;
			ELSE
				CTRL.state_axis := 20;
			END_IF
		ELSE
			TRAJ.tempo := TRAJ.tempo + TRAJ.delta_t;
		END_IF    
               
	50: // Stato 70: richiesta switch off
		CTRL.control_word	:= 0; 
		CTRL.start 		:= 0;
		CTRL.stop  		:= 0;
		CTRL.state_axis := 0;                                                                                                                                                                                                                                                                                                                                                                                                                                                                                                                                                            
END_CASE

END_PROGRAM

// ---- POUs/Trajectories/FWPoly4.TcPOU
PROGRAM FWPoly4
VAR
	a: LREAL;
	b: LREAL;
	c: LREAL;
	tempo_2: LREAL;
	tempo_3: LREAL;
	tempo_4: LREAL;
END_VAR

IF (TRAJ.tempo = 0) THEN
	TRAJ.v_max_rpm_low	:= (UDINT_TO_LREAL(TRAJ.speed_selector_rpm) / MOTOR.GEAR_RATIO);
	TRAJ.periodo_ms 	:= (ABS(TRAJ.position_selector_deg) * 15 * 1000) / (8 * TRAJ.v_max_rpm_low * 6) ; // millisecondi	
	TRAJ.delta_t 		:= 1 / (TRAJ.periodo_ms); 
	TRAJ.status			:= TRUE;
	
	a := 16 * TRAJ.v_max_rpm_low * 1000;
	b := -32 * TRAJ.v_max_rpm_low * 1000;
	c := 16 * TRAJ.v_max_rpm_low * 1000;

END_IF

IF (TRAJ.status = TRUE) THEN
	tempo_2 := TRAJ.tempo * TRAJ.tempo;
	tempo_3 := tempo_2 * TRAJ.tempo;
	tempo_4 := tempo_3 * TRAJ.tempo;
	TRAJ.target_vel_mrpm := LREAL_TO_DINT(a * tempo_4 + b * tempo_3 + c * tempo_2);
ELSE
	TRAJ.error := PLC_ERROR.TRAJ_NO_SETUP;
END_IF

END_PROGRAM

// ---- POUs/Trajectories/BWPoly4.TcPOU
PROGRAM BWPoly4
VAR
	a: LREAL;
	b: LREAL;
	c: LREAL;
	tempo_2: LREAL;
	tempo_3: LREAL;
	tempo_4: LREAL;
END_VAR

IF (TRAJ.tempo = 0) THEN
	TRAJ.v_max_rpm_low	:= (UDINT_TO_LREAL(TRAJ.speed_selector_rpm) / MOTOR.GEAR_RATIO);
	TRAJ.periodo_ms 	:= (ABS(TRAJ.position_selector_deg) * 15 * 1000) / (8 * TRAJ.v_max_rpm_low * 6) ; // millisecondi	
	TRAJ.delta_t 		:= 1 / (TRAJ.periodo_ms); 
	TRAJ.status			:= TRUE;
	
	a := -16 * TRAJ.v_max_rpm_low * 1000;
	b := 32 * TRAJ.v_max_rpm_low * 1000;
	c := -16 * TRAJ.v_max_rpm_low * 1000;

END_IF

IF (TRAJ.status = TRUE) THEN
	tempo_2 := TRAJ.tempo * TRAJ.tempo;
	tempo_3 := tempo_2 * TRAJ.tempo;
	tempo_4 := tempo_3 * TRAJ.tempo;
	TRAJ.target_vel_mrpm := LREAL_TO_DINT(a * tempo_4 + b * tempo_3 + c * tempo_2);
ELSE
	TRAJ.error := PLC_ERROR.TRAJ_NO_SETUP;
END_IF

END_PROGRAM

// ---- POUs/Modes/Cyclic_sync_torq.TcPOU
PROGRAM Cyclic_sync_torq
VAR
	timer_bool: BOOL := FALSE;
	timer_test: TON;
	back: BOOL;
END_VAR

//CYCLIC SYNC TORQUE
CASE CTRL.state_axis OF
	
    0: // State 0: Switch on request
		IF (timer_bool = FALSE) THEN
			CTRL.control_word	:= 16#6;        // Reset status
			
			timer_test(IN:=FALSE,PT:=T#3S);
			IF ((CTRL.status_word.0 = 1) AND (CTRL.status_word.4 = 1) AND (CTRL.error = 0) AND CTRL.start) THEN
				CTRL.control_word	:= 16#7;        // Switch on
				INIT();
				timer_bool := TRUE;
			END_IF
		ELSE
			IF (timer_bool)THEN
				timer_test(IN:=TRUE);
				IF ( timer_test.Q = TRUE ) THEN
					CTRL.start		:= FALSE;
					CTRL.state_axis	:= 10;
					timer_bool 		:= FALSE;  
				END_IF
			END_IF
		END_IF
	
    10:
		IF(timer_bool = FALSE) THEN
			IF ((CTRL.error = 0) AND (CTRL.status_word.1 = 1) AND (CTRL.in_opmode = MODE.CYCLIC_SYNC_TORQ)) THEN           
				TRAJ.target_torque_per_thousand	:= 0;
				CTRL.control_word := 16#0F;
				timer_test(IN:=FALSE,PT:=T#3S);
				timer_bool := TRUE;
			END_IF
		ELSE
			timer_test(IN:=TRUE);
			IF ( timer_test.Q = TRUE ) THEN
				CTRL.state_axis	:= 20;
				timer_bool	:= FALSE;  
			END_IF			
		END_IF
		
	20:
		TRAJ.target_torque_per_thousand	:= 0;
		IF ((CTRL.error = 0) AND (CTRL.in_opmode = MODE.CYCLIC_SYNC_TORQ)) THEN
			TRAJ.tempo 		:= 0;
			IF( back = TRUE) THEN
				back			:= FALSE;
				CTRL.state_axis	:= 30;
			ELSE
				back			:= TRUE;
				CTRL.state_axis	:= 40;
			END_IF
		END_IF
	
	30: 
		FWPoly3();  
		IF (TRAJ.tempo >= 1) THEN
			TRAJ.status := FALSE;
			IF (CTRL.stop) THEN
				CTRL.state_axis := 50;
			ELSE
				CTRL.state_axis := 20;
			END_IF
		ELSE
			TRAJ.tempo := TRAJ.tempo + TRAJ.delta_t;
		END_IF  
         
    40: 
		BWPoly3();
		IF (TRAJ.tempo >= 1) THEN
			TRAJ.status := FALSE;
			IF (CTRL.stop) THEN
				CTRL.state_axis := 50;
			ELSE
				CTRL.state_axis := 20;
			END_IF
		ELSE
			TRAJ.tempo := TRAJ.tempo + TRAJ.delta_t;
		END_IF    
               
	50:
		CTRL.control_word	:= 0; 
		CTRL.start 		:= 0;
		CTRL.stop  		:= 0;
		CTRL.state_axis := 0;                                                                                                                                                                                                                                                                                                                                                                                                                                                                                                                                                            
END_CASE

END_PROGRAM

// ---- POUs/Trajectories/FWPoly3.TcPOU
PROGRAM FWPoly3

VAR
	a: DINT;
	b: DINT;
	c: DINT;
	tempo_2: LREAL;
	tempo_3: LREAL;
	tempo_4: LREAL;
	torque_per_thousand: INT;
END_VAR

IF (TRAJ.tempo = 0) THEN
	TRAJ.v_max_rpm_low	:= (UDINT_TO_LREAL(TRAJ.speed_selector_rpm) / MOTOR.GEAR_RATIO);
	TRAJ.periodo_ms 	:= (ABS(TRAJ.position_selector_deg) * 15 * 1000) / (8 * TRAJ.v_max_rpm_low * 6) ; // millisecondi
	TRAJ.delta_t 		:= 1 / (TRAJ.periodo_ms); 
	TRAJ.status			:= TRUE;
	
	torque_per_thousand := LREAL_TO_INT(TRAJ.torque_selector_Nm*1000/MOTOR.RATED_TORQUE_NM);
	a := 64 * torque_per_thousand;
	b := -96 * torque_per_thousand;
	c := 32 * torque_per_thousand;

END_IF

IF (TRAJ.status = TRUE) THEN
	tempo_2 := TRAJ.tempo * TRAJ.tempo;
	tempo_3 := tempo_2 * TRAJ.tempo;
	TRAJ.target_torque_per_thousand := LREAL_TO_INT(a * tempo_3 + b * tempo_2 + c * TRAJ.tempo)/3;
ELSE
	TRAJ.error := PLC_ERROR.TRAJ_NO_SETUP;
END_IF

END_PROGRAM

// ---- POUs/Trajectories/BWPoly3.TcPOU
PROGRAM BWPoly3
VAR
	a: DINT;
	b: DINT;
	c: DINT;
	tempo_2: LREAL;
	tempo_3: LREAL;
	torque_per_thousand: DINT;
END_VAR

IF (TRAJ.tempo = 0) THEN
	TRAJ.v_max_rpm_low	:= (UDINT_TO_LREAL(TRAJ.speed_selector_rpm) / MOTOR.GEAR_RATIO);
	TRAJ.periodo_ms 	:= (ABS(TRAJ.position_selector_deg) * 15 * 1000) / (8 * TRAJ.v_max_rpm_low * 6) ; // millisecondi
	TRAJ.delta_t 		:= 1 / (TRAJ.periodo_ms); 
	TRAJ.status			:= TRUE;
	
	torque_per_thousand := LREAL_TO_INT(TRAJ.torque_selector_Nm*1000/MOTOR.RATED_TORQUE_NM);
	a := -64 * torque_per_thousand;
	b := 96 * torque_per_thousand;
	c := -32 * torque_per_thousand;

END_IF

IF (TRAJ.status = TRUE) THEN
	tempo_2 := TRAJ.tempo * TRAJ.tempo;
	tempo_3 := tempo_2 * TRAJ.tempo;
	TRAJ.target_torque_per_thousand := LREAL_TO_INT(a * tempo_3 + b * tempo_2 + c * TRAJ.tempo)/3;
ELSE
	TRAJ.error := PLC_ERROR.TRAJ_NO_SETUP;
END_IF

END_PROGRAM

// ---- DUTs/TextList.TcTLO
TEXTLIST TextList
  1 = 'Profile Position'
  3 = 'Profile Velocity'
  4 = 'Profile Torque'
  8 = 'Cyclic Sync Position'
  9 = 'Cyclic Sync Velocity'
  10 = 'Cyclic Sync Torque'
   = ''
END_TEXTLIST

// ---- GlobalTextList.TcGTLO
TEXTLIST GlobalTextList
  991 = '%.0f'
  350 = '%.1f'
  351 = '%.2f'
  669 = '%d'
  130 = '%s'
  594 = 'ACTIVE'
  274 = 'ERROR'
  461 = 'Frequency cutoff [Hz]'
  176 = 'LOADING'
  349 = 'Max speed [rpm]'
  74 = 'Motor torque [Nm]'
  405 = 'NO ETHERCAT'
  467 = 'PWR CYCLE REQ.'
  145 = 'READY'
  82 = 'RESET'
  204 = 'RESET REQUIRED'
  581 = 'SET UP'
  263 = 'Speed [rpm]'
  287 = 'START'
  209 = 'STOP'
  897 = 'Target pos [deg]'
  419 = 'Target Torque [Nm]'
  652 = 'Torque [Nm]'
  98 = 'WAITING'
END_TEXTLIST

// ---- VISUs/ControlPanel.TcVIS
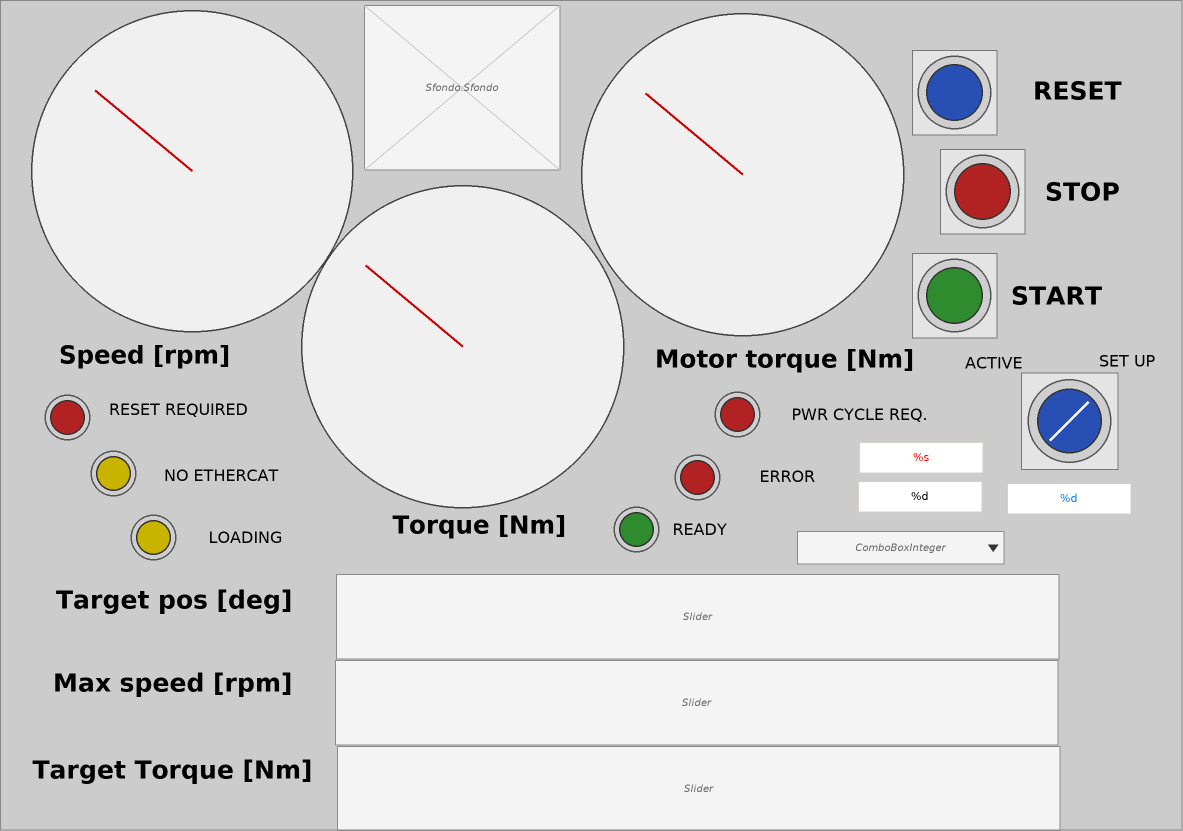
VISUALIZATION ControlPanel  // 1183x831
    Image (364,5 196x165), image: Sfondo.Sfondo
    Meter360 (300,185 325x323), value: HMI.actual_torque_nm_slow, style: Meter-Meter360-Gray, scale format: %.0f, scale -300..300
    PushSwitch (912,250 85x91), variable: CTRL.start, input disabled if: CTRL.active, behaviour: TOGGLE, style: Switch-PushSwitch-Green
    PushSwitch (937,149 91x85), variable: CTRL.stop, behaviour: TOGGLE, style: Switch-PushSwitch-Red
    Slider (335,660 723x85), variable: TRAJ.speed_selector_rpm, invisible if: CTRL.set_up, input disabled if: CTRL.set_up, scale 300..1400
    Label (31,636 284x93), "Max speed [rpm]", invisible if: CTRL.set_up
    Label (956,257 201x77), "START"
    Label (982,153 201x77), "STOP"
    Lamp1 (610,502 53x55), tooltip "WAITING", variable: CTRL.status_word.0, style: Lamp-Lamp1-Green
    Label (687,438 201x77), "ERROR"
    Label (344,502 271x46), "Torque [Nm]"
    Lamp1 (671,450 53x55), tooltip "WAITING", variable: HMI.error_light, style: Lamp-Lamp1-Red
    Label (634,491 132x77), "READY"
    Meter360 (20,10 344x322), value: HMI.actual_speed_rpm, style: Meter-Meter360-Gray, scale format: %.0f, scale -1400..1600
    Label (9,332 271x46), "Speed [rpm]"
    Meter360 (580,13 325x323), value: HMI.actual_torque_nm_fast, style: Meter-Meter360-Gray, scale format: %.1f, scale -3..3
    Label (649,336 271x46), "Motor torque [Nm]"
    PushSwitch (912,47 85x91), variable: HMI.reset_button, behaviour: TOGGLE, style: Switch-PushSwitch-Blue
    Label (977,52 201x77), "RESET"
    Lamp1 (87,446 53x55), tooltip "WAITING", variable: HMI.no_ecat_light, style: Lamp-Lamp1-Yellow
    Label (121,437 201x77), "NO ETHERCAT"
    Slider (336,574 723x85), variable: TRAJ.position_selector_deg, invisible if: CTRL.set_up, input disabled if: CTRL.set_up, scale 0..360
    Label (13,559 323x81), "Target pos [deg]", invisible if: CTRL.set_up
    ComboBoxInteger (797,531 207x33), variable: CTRL.opmode, input disabled if: CTRL.set_up, text list: 'TextList'
    Slider (337,746 723x85), variable: TRAJ.torque_selector_Nm, invisible if: CTRL.set_up, input disabled if: CTRL.set_up, scale 0..5
    Label (18,724 309x91), "Target Torque [Nm]", invisible if: CTRL.set_up
    Lamp1 (41,390 53x55), tooltip "WAITING", variable: HMI.reset_light, style: Lamp-Lamp1-Red
    Label (78,371 201x77), "RESET REQUIRED"
    Lamp1 (711,387 53x55), tooltip "WAITING", variable: HMI.out_limits_light, style: Lamp-Lamp1-Red
    Label (749,376 221x77), "PWR CYCLE REQ."
    Textfield (859,442 124x31), "%s", text variable: SDO.error_report
    RotarySwitch (1021,369 97x104), variable: CTRL.set_up, input disabled if: CTRL.wait, behaviour: TOGGLE, style: Switch-RotarySwitch-Blue
    Label (958,329 72x68), "ACTIVE"
    Label (1088,327 78x68), "SET UP"
    Lamp1 (127,510 53x55), tooltip "WAITING", variable: CTRL.wait, style: Lamp-Lamp1-Yellow
    Label (156,499 179x77), "LOADING"
    Textfield (1007,483 124x31), "%d", text variable: CTRL.status_word
    Textfield (858,481 124x31), "%d", text variable: CTRL.state_axis
END_VISUALIZATION
